INTERFACE I_Valve

PROPERTY Error : BOOL
GET
END_GET
SET
END_SET
END_PROPERTY

PROPERTY OpeningActual : REAL
GET
END_GET
SET
END_SET
END_PROPERTY

PROPERTY OpeningSetpoint : REAL
GET
END_GET
SET
END_SET
END_PROPERTY

METHOD Run
VAR_INPUT
END_VAR
END_METHOD

END_INTERFACE

(* stored: Version 1.1.0.1, ProductVersion 3.1.4024.0
   Itf I_Valve: Id {4cab4434-0ff2-463c-97d2-f53a68202f0c}
   Property Error: Id {86a70818-06b2-47a6-9e69-4d16243b0647}
   Get Get: Id {41ea2990-43cc-4e51-8cb0-2213c484ddcc}
   Set Set: Id {547892e8-2b81-4095-8e60-79c061a964c7}
   Property OpeningActual: Id {f78afc7a-c45b-4606-9d33-64d307f40524}
   Get Get: Id {ff6cce24-ddbc-423d-9108-08fb867a819b}
   Set Set: Id {4fead4e0-ccdd-4903-9e7c-a61473ede478}
   Property OpeningSetpoint: Id {64ee94a4-7af2-40f1-87be-5fc9dfbc99df}
   Get Get: Id {27ca2882-4156-4781-aef3-5f7f4e12ba13}
   Set Set: Id {adc15932-790f-4bc7-b5f0-96902ebc8d9b}
   Method Run: Id {af639dba-9bd2-40ad-bf55-1ad6e0146b5d} *)
